// TIA Portal V19 export
FUNCTION "CT DOSING" : Void   // FC95, STL
{ S7_Optimized_Access := 'TRUE' }
AUTHOR : OPA_8160
FAMILY : OPTION
NAME : CT_DOSIN
VERSION : 0.0
// THIS FUNCTION BLOCK SHOULD ONLY BE USED IF THE ASEPTIC TANK HAS ITS OWN 
// LYE/ACID-CONTAINERS AND CONDUCTIVITY METER. THE FUNCTION BLOCK BEHAVE 
// JUST LIKE THE UHT WOULD HAVE RESPONDED ON LYE/ACID REQUESTS, BUT DOSING 
// TIMERS HAS TO BE REPLACED WITH "CT LYE OK" AND "CT ACID OK" IN THE CIP
// PROGRAM. PLEASE BE AWARE THAT "CT LYE OK" AND "CT ACID OK" HAS TO BE RESET
// IN THE CIP PROGRAM AS WELL.
// SOFTWARE SIMULATED IN OFFICE 10/2 1998  
// 
// ****** REVISION HISTORY :
// 
// VERSION DATE         BY    DESCRIPTION
// --------------------------------------------------------------------------
// 00.00     9/2 1997   OPA   ORIGINAL FUNCTION BLOCK CREATED
//       
// 00.01    17/8 2000   BUG   Load setpoint when filler in CIP
// stored: AutoNumber false
   VAR_TEMP
      Temp_Lye : Real;
      Temp_Acid : Real;
   END_VAR
BEGIN

NETWORK
TITLE = DOSING LYE/ACID
      A     "S0 FILLER";
      JC    FSP;  // FSP Jump to filler setpoint
      L     "Setpoints".CT2073LyeConcSpCIP;  // Load Tank Setpoint
      T     #Temp_Lye;
      L     "Setpoints".CT2073AcidConcSpCIP;
      T     #Temp_Acid;
      JU    Con;

FSP:  L     "Setpoints".CT2073LyeConcSpFiller;  // Load Filler Setpoint
      T     #Temp_Lye;
      L     "Setpoints".CT2073AcidConcSpFiller;
      T     #Temp_Acid;

Con:  A     "Continue_in program";
      S     "TIM54";
      S     "TIM55";
      S     "ProcessAndPbAlarms"."A"[17];  //A17_ContinueDosingSelect// Event
      R     "Continue_in program";
      BEC;

      AN    "TANK AUTO";
      AN    "S0 FILLER";  // add by bug, acid dos always start with alarm ?
      AN    "S.T.01.REQUEST LYE";
      AN    "S.T.01.REQUEST ACID";
      BEC;
      O     "S.T.01.REQUEST LYE";
      O     "S.T.01.REQUEST ACID";
      JC    mx;
      R     "MY0237";
      R     "MY0238";
      R     "T54 LYE DOSING TOO LONG";
      R     "T55 ACID DOSING TOO LONG";
      R     "R.CIP UNIT OCCUPIED";
      R     "Dummy Start CIP timer";
      BEU;
mx:   A     "Dummy Start CIP timer";
      JC    M002;
      S     "TIM54";
      S     "TIM55";
      S     "Dummy Start CIP timer";

M002: A     "R.CIP UNIT OCCUPIED";
      JC    M003;
      S     "R.CIP UNIT OCCUPIED";
//      S     "TIM54"                     // SET SECURITY TIMER FOR DOSING LYE
//      S     "TIM55"                     // SET SECURITY TIMER FOR DOSING ACID
      BEU;
M003: NOP   0;

NETWORK
TITLE = CALCULATE ALLOWED DEVIATION FROM SETPOINT
// L     1.000000e+002
//       L     "DB SETPOINTS".CT2073MaxDeviationConcSp
//       -R    
//       L     1.000000e+002
//       /R    
//       T     "DB SETPOINTS".CalculationLowLimit
// 
//       L     1.000000e+002
//       L     "DB SETPOINTS".CT2073MaxDeviationConcSp
//       +R    
//       L     1.000000e+002
//       /R    
//       T     "DB SETPOINTS".CalculationHighLimit

NETWORK
TITLE = DOSE LYE UNTIL CONCENTRATION IS WITHIN LIMITS
      A     "S.T.01.REQUEST LYE";
      JC    c007;
      JC    END;
c007: AN    "T54 LYE DOSING TOO LONG";
      S     "ProcessAndPbAlarms"."A"[40];  //A40_LyedosingTooLong//ALARM "LYE DOSING TOO LONG"
//      A     "B02.76"                    //LYE CONTAINER EMPTY
      A     "R.Lye Level Ok";
      JC    c008;
      S     "ProcessAndPbAlarms"."A"[46];  //A46_LyeContainerEmpty//ALARM LYE CONTAINER EMPTY
c008: L     #Temp_Lye;  // Lye Setpoint
      L     "MeasuredValues".CT0182REAL;  //"DB-ANALOG INPUT".CT0182REAL    // ANALOG CONDUCTIVITY METER INPUT
      >R;  // CONDUCTIVITY < SETPOINT-DEVIATION
      A     "T54 LYE DOSING TOO LONG";
      S     "MY0237";  // START LYE DOSING
      R     "T53 DETERGENT CONC OK";  // RESET TIMER LYE CONC OK
      BEC;
      AN    "T54 LYE DOSING TOO LONG";
      R     "MY0237";
      BEC;
// IF SECURITY DOSING TIMER EXPIRES, THEN GIVE ALARM AND CONTINUE DOSING
// "AGREEMENT WITH WOLFGANG, UNIT SYSTEMS", THE SAME METHOD AS UHT CLESA SPAIN
// CHANGED BY - POS - 05.07.2000. AGREEMENT WITH BESTFOOD.
      AN    "MY0237";
      AN    "T53 DETERGENT CONC OK";  // TIMER LYE CONC OK
      S     "CT_LYE_OK";  // CT LYE OK

      L     #Temp_Lye;  // Lye Setpoint
      L     "MeasuredValues".CT0182REAL;  // "DB-ANALOG INPUT".CT0182REAL    // ANALOG CONDUCTIVITY METER INPUT
      <R;  // CONDUCTIVITY > SETPOINT+DEVIATION
      A     "MY0237";
      S     "TIM53";  // START TIMER LYE CONC OK
      R     "MY0237";  // RESET LYE DOSING
      BEU;
END:  NOP   0;

NETWORK
TITLE = DOSE LYE UNTIL CONCENTRATION IS WITHIN LIMITS
      A     "S.T.01.REQUEST ACID";
      JC    c009;
      JC    END1;
c009: AN    "T55 ACID DOSING TOO LONG";
      S     "ProcessAndPbAlarms"."A"[41];  //A41_AcidDosingTooLong//ALARM "ACID DOSING TOO LONG"
//      A     "B02.77"                    //ACID CONTAINER EMPTY
      A     "R.Acid Level Ok";
      JC    c010;
      S     "ProcessAndPbAlarms"."A"[47];  //A47_AcidContainerEmpty//ALARM ACID CONTAINER EMPTY
c010: L     #Temp_Acid;  // Acid Setpoint
      L     "MeasuredValues".CT0182REAL;  //"DB-ANALOG INPUT".CT0182REAL    // ANALOG CONDUCTIVITY METER INPUT
      >R;  // CONDUCTIVITY < SETPOINT-DEVIATION
      A     "T55 ACID DOSING TOO LONG";
      S     "MY0238";  // START ACID DOSING
      R     "T53 DETERGENT CONC OK";  // RESET TIMER ACID CONC OK
      BEC;
      AN    "T55 ACID DOSING TOO LONG";
      R     "MY0238";
      BEC;
// IF SECURITY DOSING TIMER EXPIRES, THEN GIVE ALARM AND CONTINUE DOSING
// "AGREEMENT WITH WOLFGANG, UNIT SYSTEMS", THE SAME METHOD AS UHT CLESA SPAIN
// CHANGED BY - POS - 05.07.2000. AGREEMENT WITH BESTFOOD.
      AN    "MY0238";
      AN    "T53 DETERGENT CONC OK";  // TIMER ACID CONC OK
      S     "CT_ACID_OK";  // CT ACID OK

      L     #Temp_Acid;  // Acid Setpoint
      L     "MeasuredValues".CT0182REAL;  //"DB-ANALOG INPUT".CT0182REAL    // ANALOG CONDUCTIVITY METER INPUT
      <R;  // CONDUCTIVITY > SETPOINT+DEVIATION
      A     "MY0238";
      S     "TIM53";  // START TIMER ACID CONC OK
      R     "MY0238";  // RESET ACID DOSING
      BEU;
END1: NOP   0;
END_FUNCTION
